TYPE ST_AddCommand EXTENDS ST_BasicCommand :
STRUCT
	stArgsIn		: ST_AddCommandIn;
	stArgsOut		: ST_AddCommandOut;
END_STRUCT
END_TYPE

(* stored: Version 1.1.0.1, ProductVersion 3.1.4022.9
   DUT ST_AddCommand: Id {dbec02be-ef92-4686-830f-a6cf180a80a0} *)
